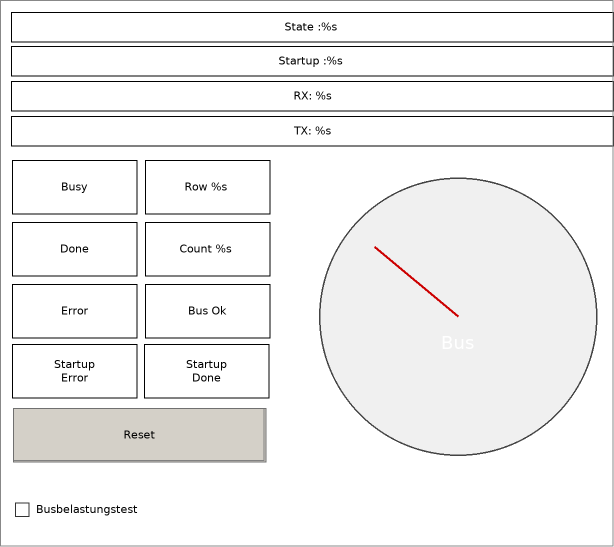
VISUALIZATION BusRS485Master_Frame_1  // 614x547
VAR_IN_OUT	
	(* für RS485 FiFo Master *)
	bBusBelastungstest		:BOOL;
	bReset					:BOOL;
	
	stFiFoMasterState		:ST_FiFoMaster_State;
	stRS48StartupState		:ST_RS485Startup_State;
END_VAR
    Meter360 (319,170 278x293), value: stFiFoMasterState.lrBusAuslastung, style: Meter-Meter360-Gray, scale format: %.1f, scale 0..350
    Rectangle (11,81 603x30), "RX: %s", text variable: stFiFoMasterState.sReceiveString
    Checkbox (13,472 254x75), "Busbelastungstest", variable: bBusBelastungstest
    Rectangle (11,116 603x30), "TX: %s", text variable: stFiFoMasterState.sSendString
    Rectangle (11,12 603x30), "State :%s", text variable: stFiFoMasterState.sState
    Rectangle (12,160 125x54), "Busy", colour toggle: stFiFoMasterState.bBusy
    Rectangle (12,222 125x54), "Done", colour toggle: stFiFoMasterState.bDone
    Rectangle (12,284 125x54), "Error", colour toggle: stFiFoMasterState.bError
    Rectangle (145,160 125x54), "Row %s", text variable: stFiFoMasterState.iFiFoRow
    Rectangle (145,222 125x54), "Count %s", text variable: stFiFoMasterState.iFiFoCount
    Button (13,408 253x54), "Reset"
        tap bReset
    Label (383,328 150x30), "Bus"
    Rectangle (11,46 603x30), "Startup :%s", text variable: stRS48StartupState.sStartupState
    Rectangle (145,284 125x54), "Bus Ok", colour toggle: stRS48StartupState.bBusOk
    Rectangle (144,344 125x54), "Startup Done", colour toggle: stRS48StartupState.bStartupDone
    Rectangle (12,344 125x54), "Startup Error", colour toggle: stRS48StartupState.bStartupError
END_VISUALIZATION

(* stored: Version 1.1.0.1, ProductVersion 3.1.4024.12
   Visu BusRS485Master_Frame_1: Id {81e195db-d6dd-4c40-b668-8ff45670e61b} *)
